RoboDK station: SelfFoundStation.rdk

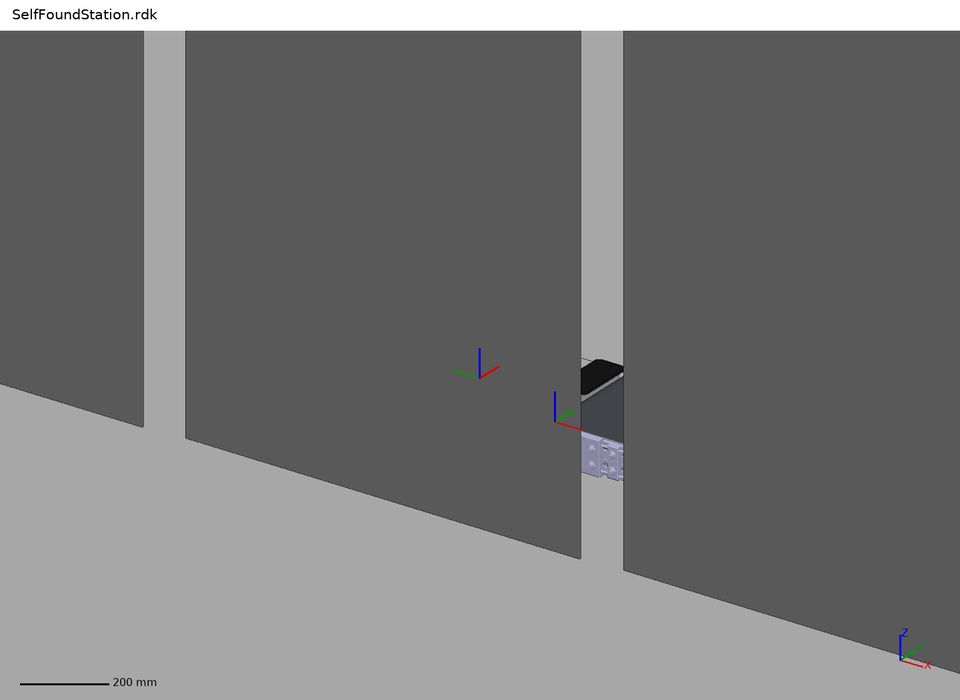
[picture v0: the station drawn from its stored meshes, robots at their saved joint values, targets as dots, program paths as lines]
Station SelfFoundStation (saved by RoboDK 5.7.4). Poses are relative to the parent item; angles as X-Y-Z fixed-axis rotations.
  - Python program ImportCode (listed below)
  - Python program ResetCode (listed below)
  - Python program ResetPositionCode (listed below)
  - Python program MainProg (listed below)
  - frame MAIN Base at (0, 1000, 0) mm
    - frame Dobot Magician Base at (-1020, -980, 50) mm, rotated rx 0 ry 0 rz 90 deg
      - robot Dobot Magician: 4 axes, payload 0.5 kg, reach 320 mm, repeatability 0.2 mm, weight 4 kg
          joint limits [-90, -0.001, -10, -90] to [90, 85, 95, 90]; home [0, 0, 0, 0]; saved at [0, 0, 0, 0]
        - tool Tool1, TCP at (0, 0, 117.4) mm, size 100 x 100 x 114.9 mm
    - frame CON1 Base at (-660, -1200, 130) mm
      - robot CON1: 1 axes
          modified DH rows (alpha deg, a mm, theta deg, d mm): 0, 0, 0, 0 linear
          base shift (0, 0, 0) mm, rotated rx 0 ry 90 rz 0 deg
          joint limits [-500000] to [500000]; home [0]; saved at [-1980]
        - object Item at (1930, 230, 0) mm, rotated rx -90 ry 0 rz 0 deg, size 78.4 x 12 x 160.7 mm, geometry from Item.stl
    - object Room at (0, 0, 0) mm, size 10000 x 10000 x 25 mm, geometry from Room.stl
    - object Panels at (-2000, 0, 0) mm, size 5655.1 x 3636 x 2268 mm, geometry from Panels.sld
    - object Table at (-810, -980, 0) mm, size 200 x 200 x 120 mm, geometry from Table.stl
    - object Warehouse at (-1330, -980, 20) mm, rotated rx 0 ry 0 rz 90 deg, size 400 x 400 x 50 mm, geometry from Warehouse.stl

--- Python program ImportCode ---
from robodk import robolink    # RoboDK API
from robodk import robomath    # Robot toolbox
from robodk import * # RoboDK API
from robodk.robolink import * # RoboDK API

RDK = robolink.Robolink()

# ----------------------------------------------------------------
# 1. 최상위 프레임 생성
# ----------------------------------------------------------------
def ADDFrame():
    # 모든 요소의 기준이 될 메인 베이스 하나만 깔끔하게 생성합니다.
    MAIN_Base = RDK.AddFrame("MAIN Base")
    return MAIN_Base


# ----------------------------------------------------------------
# 2. 로봇 및 오브젝트 로드 함수
# ----------------------------------------------------------------
def addfile_robot(main_base):
    # 로봇 자체 베이스가 생성되므로 main_base 바로 아래에 로드합니다.
    dobot_item = RDK.AddFile(r'C:\work\SelfFound\roboDK\Dobot-Magician.robot', main_base)

    # 자동으로 생성된 로봇 프레임의 이름을 우리가 원하는 형태로 변경하여 중복을 방지합니다.
    # 트리에서 생성된 고유 프레임 객체를 찾아 이름을 강제로 세팅합니다.
    dobot_base_frame = RDK.Item("Dobot Magician Base", 3)
    if not dobot_base_frame.Valid():
        # 만약 로봇 기본 이름으로 프레임이 생성되었다면 찾아서 이름을 변경
        auto_frame = RDK.Item("Dobot-Magician Base", 3)
        if auto_frame.Valid():
            auto_frame.setName("Dobot Magician Base")


def addfile_tool():
    # 💡 [수정] 변경된 로봇 이름을 정확히 추적할 수 있도록 예외 처리를 추가합니다.
    robot_item = RDK.Item("Dobot Magician", 2)
    if not robot_item.Valid():
        robot_item = RDK.Item("Dobot-Magician", 2)

    if robot_item.Valid():
        RDK.AddFile(r'C:\work\SelfFound\roboDK\Tool1.tool', robot_item)


def addfile_conveyor(main_base):
    # 컨베이어 벨트도 자동으로 베이스가 생기므로 main_base 바로 아래에 로드합니다.
    con1_item = RDK.AddFile(r'C:\work\SelfFound\roboDK\CON1.robot', main_base)

    # 자동으로 생성된 컨베이어 베이스 프레임 이름 정렬
    con1_base_frame = RDK.Item("CON1 Base", 3)
    if not con1_base_frame.Valid():
        auto_frame = RDK.Item("CON1 Base", 3)
        if auto_frame.Valid():
            auto_frame.setName("CON1 Base")


def addfile_object(main_base):
    # 💡 [수정] 중복 로드되던 warehouse.sld를 제거하고 정확한 파일 목록만 정렬합니다.
    RDK.AddFile(r'C:\work\SelfFound\roboDK\Room.stl', main_base)
    RDK.AddFile(r'C:\work\SelfFound\roboDK\Panels.sld', main_base)
    RDK.AddFile(r'C:\work\SelfFound\roboDK\Table.stl', main_base)
    RDK.AddFile(r'C:\work\SelfFound\roboDK\Warehouse.stl', main_base)
    RDK.AddFile(r'C:\work\SelfFound\roboDK\Item.stl', main_base)


# ----------------------------------------------------------------
# 3. 메인 실행 제어
# ----------------------------------------------------------------
# 1) 기준점이 되는 MAIN Base 프레임을 하나 만듭니다.
main_b = ADDFrame()

# 2) 중복 프레임이 발생하지 않도록 각 함수에서 이름을 제어하며 에셋들을 로드합니다.
addfile_robot(main_b)
addfile_tool()
addfile_conveyor(main_b)
addfile_object(main_b)

--- Python program ResetCode ---
from robodk import robolink    # RoboDK API
from robodk import robomath    # Robot toolbox
RDK = robolink.Robolink()
from robodk import * # RoboDK API
from robodk.robolink import * # Robot toolbox
# Link to RoboDK


#로봇 선언
Dobot=RDK.Item("Dobot-Magician", 2)
if not Dobot.Valid():
    Dobot=RDK.Item("Dobot Magician", 2)
CON1=RDK.Item("CON1", 2)

#오브젝트 선언
Room=RDK.Item("Room", 5)
Panels=RDK.Item("Panels", 5)
Warehouse=RDK.Item("Warehouse", 5)
Table=RDK.Item("Table", 5)
Item_Object=RDK.Item("Item", 5)

#Tool 선언
Tool1=RDK.Item("Tool1", 4)

#프레임 선언
MAIN_Base=RDK.Item("MAIN Base", 3)
Dobot_Base=RDK.Item("Dobot Magician Base", 3)
if not Dobot_Base.Valid():
    Dobot_Base=RDK.Item("Dobot-Magician Base", 3)
CON1_Base=RDK.Item("CON1 Base", 3)


# ----------------------------------------------------------------
# 이미지 트리 창 기준 최종 계층 구조 정의
# ----------------------------------------------------------------

# 1) 베이스 프레임들을 MAIN Base 하위로 종속
if Dobot_Base.Valid() and MAIN_Base.Valid(): Dobot_Base.setParent(MAIN_Base)
if CON1_Base.Valid() and MAIN_Base.Valid(): CON1_Base.setParent(MAIN_Base)

# 2) 도봇 로봇 본체와 툴 구조 조립
if Dobot.Valid() and Dobot_Base.Valid(): Dobot.setParent(Dobot_Base)
if Tool1.Valid() and Dobot.Valid(): Tool1.setParent(Dobot)

# 3) 컨베이어 벨트 본체를 CON1 Base 하위로 종속
if CON1.Valid() and CON1_Base.Valid(): CON1.setParent(CON1_Base)

# 4) 💡 요청하신 사항: Item이 CON1(컨베이어 장치)을 부모로 따라가도록 묶기
if Item_Object.Valid() and CON1.Valid():
    Item_Object.setParent(CON1)

# 5) 나머지 환경 및 적재 오브젝트들은 MAIN Base 하위로 일렬 정렬
if Room.Valid() and MAIN_Base.Valid(): Room.setParent(MAIN_Base)
if Panels.Valid() and MAIN_Base.Valid(): Panels.setParent(MAIN_Base)
if Table.Valid() and MAIN_Base.Valid(): Table.setParent(MAIN_Base)
if Warehouse.Valid() and MAIN_Base.Valid(): Warehouse.setParent(MAIN_Base)

print("이미지 트리 기준 구조 조립 및 Item-컨베이어 부모 결합이 완료되었습니다.")

--- Python program ResetPositionCode ---
from robodk import robolink    # RoboDK API
from robodk import robomath    # Robot toolbox
from robodk import * # RoboDK API
from robodk.robolink import * # RoboDK API

RDK = robolink.Robolink()

# ----------------------------------------------------------------
# 1. 트리 창에 존재하는 실제 아이템 객체 정의
# ----------------------------------------------------------------
MAIN_Base = RDK.Item("MAIN Base", 3)
Dobot_Base = RDK.Item("Dobot Magician Base", 3)
CON1_Base = RDK.Item("CON1 Base", 3)

Dobot = RDK.Item("Dobot-Magician", 2)
CON1 = RDK.Item("CON1", 2)

Room = RDK.Item("Room", 5)
Panels = RDK.Item("Panels", 5)
Warehouse = RDK.Item("warehouse", 5)

Table = RDK.Item("Table", 5)
Warehouse = RDK.Item("Warehouse", 5)
Item = RDK.Item("Item", 5)


# ----------------------------------------------------------------
# 2. 설계도 기반 정밀 좌표 재배치 (단위: mm)
# ----------------------------------------------------------------

Panels.setPose(Mat([[     1.000000,     0.000000,     0.000000, -2000.000000 ],
      [     0.000000,     1.000000,     0.000000,     0.000000 ],
      [     0.000000,     0.000000,     1.000000,     0.000000 ],
      [     0.000000,     0.000000,     0.000000,     1.000000 ]]))

CON1_Base.setPose(Mat([[     1.000000,     0.000000,     0.000000,  -660.000000 ],
      [     0.000000,     1.000000,     0.000000, -1200.000000 ],
      [     0.000000,     0.000000,     1.000000,   130.000000 ],
      [     0.000000,     0.000000,     0.000000,     1.000000 ]]))

# Table
Table.setPose(Mat([[     1.000000,     0.000000,     0.000000,  -810.000000 ],
      [     0.000000,     1.000000,     0.000000, -980.000000 ],
      [     0.000000,     0.000000,     1.000000,     0.000000 ],
      [     0.000000,     0.000000,     0.000000,     1.000000 ]]))

# 💡 도봇의 정면이 화면 위쪽(북쪽)을 바라보도록 회전 성분을 수정했습니다.
Dobot_Base.setPose(Mat([[     0.000000,    -1.000000,     0.000000, -1020.000000 ],
      [     1.000000,     0.000000,     0.000000, -980.000000 ],
      [     0.000000,     0.000000,     1.000000,     50.000000 ],
      [     0.000000,     0.000000,     0.000000,     1.000000 ]]))

# warehouse
Warehouse.setPose(Mat([[     0.000000,    -1.000000,     0.000000, -1330.000000 ],
      [     1.000000,     0.000000,     0.000000, -980.000000 ],
      [     0.000000,     0.000000,     1.000000,    20.000000 ],
      [     0.000000,     0.000000,     0.000000,     1.000000 ]]))

# lost_item
Item.setPose(Mat([[     1.000000,    0.000000,     0.000000,  1930.000000 ],
      [     0.000000,     0.000000,     1.000000, 230.000000 ],
      [     0.000000,     -1.000000,     0.000000,   0.000000 ],
      [     0.000000,     0.000000,     0.000000,     1.000000 ]]))



# ----------------------------------------------------------------
# 3. 내부 장치 및 관절각 초기화
# ----------------------------------------------------------------
if CON1.Valid():
    CON1.setPose(Mat([[1, 0, 0, 0], [0, 1, 0, 0], [0, 0, 1, 0], [0, 0, 0, 1]]))

if Dobot.Valid():
    Dobot.setPose(Mat([[1, 0, 0, 0], [0, 1, 0, 0], [0, 0, 1, 0], [0, 0, 0, 1]]))
    Dobot.MoveJ([0, 0, 45, 45, 0])

print("설계도 흐름에 맞추어 좌우 축 반전 정밀 재배치가 완료되었습니다.")

--- Python program MainProg ---
from robodk import robolink    # RoboDK API
from robodk import robomath    # Robot toolbox
RDK = robolink.Robolink()
from robodk import * # RoboDK API
from robolink import * # Robot toolbox
import time

#로봇 선언
Dobot=RDK.Item("Dobot-Magician", 2)
if not Dobot.Valid():
    Dobot=RDK.Item("Dobot Magician", 2)
CON1=RDK.Item("CON1", 2)

#오브젝트 선언
Room=RDK.Item("Room", 5)
Panels=RDK.Item("Panels", 5)
Warehouse=RDK.Item("Warehouse", 5)
Table=RDK.Item("Table", 5)
Item_Object=RDK.Item("Item", 5)

#Tool 선언
Tool1=RDK.Item("Tool1", 4)

#프레임 선언
MAIN_Base=RDK.Item("MAIN Base", 3)
Dobot_Base=RDK.Item("Dobot Magician Base", 3)
if not Dobot_Base.Valid():
    Dobot_Base=RDK.Item("Dobot-Magician Base", 3)
CON1_Base=RDK.Item("CON1 Base", 3)


# ----------------------------------------------------------------
# 1. 컨베이어 이송 구동 함수 (생략)
# ----------------------------------------------------------------
def job1_conveyor():
    print("컨베이어 마이너스 방향 이송을 시작합니다.")
    for x_pos in range(-540, -2000, -20):
        if CON1.Valid():
            CON1.setPose(transl(x_pos, 0.0, 0.0))
            RDK.Render()
            time.sleep(0.02)
    print("컨베이어 이송 완료.")


# ----------------------------------------------------------------
# 2. 도봇 매지션 흡착 및 Warehouse 이송 함수 (도달 반경 오프셋 보정)
# ----------------------------------------------------------------
def job2_dobot_pick_and_place():
    print("도봇 피크 앤 플레이스 시작...")

    if Dobot.Valid() and Table.Valid() and Warehouse.Valid() and Dobot_Base.Valid():
        # 도봇의 좌표 기준 프레임 설정
        Dobot.setPoseFrame(Dobot_Base)

        # 💡 [조율 포인트 1] Table 중심점 기준 도봇이 닿을 수 있는 물리 반경으로 보정
        # 테이블의 원점 위치에서 도봇 팔이 도달 가능한 범위로 transl(X, Y, Z) 수치를 깎아줍니다.
        # 에러가 나면 도봇 몸체 쪽으로 오도록 값을 더하거나 빼며 튜닝해야 합니다.
        table_matrix = Table.Pose()
        target_pos = invH(Dobot_Base.Pose()) * table_matrix * transl(0, 0, 120)

        # Table 상단 공중으로 이동 시도
        Dobot.MoveJ(target_pos)
        Dobot.MoveL(Dobot.Pose() * transl(0, 0, -120))  # 물건 밀착 하강

        # 진공 흡착(Vaccum ON) 작동
        Tool1.AttachClosest("Item", 2000)

        # 안전 높이로 위로 들어 올리기
        Dobot.MoveL(Dobot.Pose() * transl(0, 0, 100))

        # 💡 [조율 포인트 2] Warehouse 중심점 기준 도봇 도달 범위 보정
        warehouse_matrix = Warehouse.Pose()
        warehouse_target = invH(Dobot_Base.Pose()) * warehouse_matrix * transl(0, 0, 100)

        # Warehouse 상단으로 이동 후 적재 위치로 하강
        Dobot.MoveJ(warehouse_target)
        Dobot.MoveL(Dobot.Pose() * transl(0, 0, -100))

        # 진공 해제(Vaccum OFF)
        Tool1.DetachAll(MAIN_Base)

        # 로봇 팔 안전 회피 상승
        Dobot.MoveL(Dobot.Pose() * transl(0, 0, 100))


# ----------------------------------------------------------------
# 3. 도봇 복귀 및 초기 방향(북쪽) 정렬 함수
# ----------------------------------------------------------------
def job3_return_home():
    if Dobot.Valid():
        Dobot.MoveJ([0, 0, 45, 45, 0])


# ----------------------------------------------------------------
# 메인 프로세스 시퀀스 실행
# ----------------------------------------------------------------
job1_conveyor()
job2_dobot_pick_and_place()
job3_return_home()
